// TwinCAT 3 PLC project Nepionic_Log_Klein
// Title: Nepionic_Log_Klein
// Company: Nepionic
// Author: Nepionic
// ProjectVersion: 0.1.0
// ProgramVersion: 3.1.4026.22
// libraries:
//   [Nepionic_Log], * (Nepionic)
//   Tc2_System, * (Beckhoff Automation GmbH)
//   Tc2_Utilities, * (Beckhoff Automation GmbH)
// project tree:
//   Lib/ KleinEventAppender.TcPOU, KleinEventEntry.TcDUT, KleinEventRing.TcDUT

// ---- Lib/KleinEventEntry.TcDUT
// One slot in the KleinEventRing.
//
// Binary layout (1280 bytes, little-endian, IDENTICAL in shape to
// Nepionic_Log_OTel.OTelLogEntry — see that type's doc comment. This is a
// deliberate reuse of the same proven wire layout under a new type name, not
// a coincidence: there is no reason to invent a different byte layout when
// this one is already implemented, tested, and documented on the Go side
// (github.com/siyka-au/klein, internal/receiver/ads/eventring.go). Giving it
// its own type name (rather than literally reusing OTelLogEntry) makes it an
// independently addressable ADS symbol under Nepionic_Log_Klein, decoupled
// from the deprecated Nepionic_Log_OTel library.
//
//   offset    0  ULINT   timestamp         Unix epoch nanoseconds
//   offset    8  UDINT   severity          0=Debug 1=Info 2=Warning 3=Error 4=Fatal
//                                            (raw PLC LogLevel ordinal — see the
//                                            PLC LogLevel -> Klein Severity mapping below)
//   offset   12  UDINT   attr_count        Number of populated entries in attrs (0..10)
//   offset   16  BYTE[192] message         STRING(191) null-terminated
//   offset  208  BYTE[64]  source          STRING(63)  null-terminated (instance path)
//   offset  272  BYTE[960] attrs           ARRAY[0..9] OF Nepionic_Log.LogAttribute (96 bytes each)
//                                            each attr:
//                                              offset  0  key         STRING(31)       = 32 bytes
//                                              offset 32  attr_type   LogAttributeType =  1 byte
//                                              offset 33  value_bytes ARRAY[0..62]     = 63 bytes
//   offset 1232  BYTE[44]  _pad
//   offset 1276  UDINT   sequence          ODD=being written, EVEN=committed (LAST field)
//   Total: 1280 bytes
//
// --- PLC LogLevel -> Klein Event mapping (Go: internal/receiver/ads/eventring.go) ---
//
// This is the precise mapping the Go decoder (KleinEventEntry -> model.Event)
// implements, documented here since no PLC toolchain was available in the
// authoring environment to verify it end-to-end against a live ring:
//
//   severity (raw UDINT, PLC LogLevel ordinal) -> model.Severity (klein/internal/model.Event.go):
//     0 (Debug)       -> SeverityDebug (2)
//     1 (Information) -> SeverityInfo  (3)
//     2 (Warning)     -> SeverityWarn  (4)
//     3 (Error)       -> SeverityError (5)
//     4 (Fatal)       -> SeverityFatal (6)
//     anything else   -> SeverityInfo  (3), clamped/defaulted (out-of-range raw value)
//
//   message   -> Event.Message                       (verbatim)
//   source    -> Event.Signal.Path                    (the resulting Event's identity)
//   source    -> Event.Actor.ID, with Event.Actor.Type fixed to "plc"
//               (a PLC-origin Event always carries a fixed Actor{Type: "plc", ID: source})
//   attrs[0..attr_count-1]
//             -> Event.To, as a model.StructValue{Fields: {attr.key: attr.value, ...}}
//                only when attr_count > 0 — an Event with no attributes leaves To nil
//                rather than emitting an empty Struct (Event has no dedicated
//                attributes field; To/From are otherwise unused by a pure
//                log-message Event, per docs/SPEC.md §9's "context lives either
//                as extra fields inside value's Struct, or in the sibling
//                attributes map" convention, adapted here since Event has no
//                sibling attributes map of its own).
//   timestamp -> Event.SourceTimestamp (int64 ns, direct copy)
{attribute 'pack_mode' := '1'}
TYPE KleinEventEntry :
STRUCT
	timestamp : ULINT;
	severity : UDINT;
	attribute_count : UDINT(0..10);
	message : STRING(191);
	source : STRING(63);
	attributes : ARRAY[0..9] OF Nepionic_Log.LogAttribute;
	_pad : ARRAY[0..43] OF BYTE;
	sequence : UDINT;
END_STRUCT
END_TYPE

// ---- Lib/KleinEventRing.TcDUT
// Ring buffer header + 128-slot event entry array.
// Exposed as an ADS symbol (e.g. MAIN.klein_appender.ring) and read by the Go
// Klein collector's ADS receiver (github.com/siyka-au/klein,
// internal/receiver/ads/eventring.go — DrainEvents/ParseEventSlot).
//
// Binary layout — IDENTICAL in shape to Nepionic_Log_OTel.OTelLogRing (same
// 64-byte header, same 128 x 1280-byte entries array). Deliberately reusing
// the proven ring-header layout under a new type name; see KleinEventEntry's
// doc comment for why.
//
//   offset  0  UDINT  head          Monotonically increasing write counter
//   offset  4  UDINT  capacity      Number of slots = 128
//   offset  8  UDINT  overflow_cnt  Incremented when ring is full
//   offset 12  UDINT  _reserved
//   offset 16  BYTE[48] _cache_pad  Pad header to 64 bytes
//   offset 64  KleinEventEntry[128] 128 x 1280 bytes = 163840 bytes
//   Total: 163904 bytes
TYPE KleinEventRing :
STRUCT
	head : UDINT;
	capacity : UDINT := 128;
	overflow_cnt : UDINT;
	_reserved : UDINT;
	_cache_pad : ARRAY[0..47] OF BYTE;
	entries : ARRAY[0..127] OF KleinEventEntry;
END_STRUCT
END_TYPE

// ---- Lib/KleinEventAppender.TcPOU
{attribute 'linkalways'}
{attribute 'no_explicit_call' := 'This FB is a CLASS and must be accessed using methods or properties'}
{attribute 'enable_dynamic_creation'}
/// Klein Event appender for Nepionic_Log.
/// Implements `LogAppender` by writing structured log entries directly into its
/// own `KleinEventRing` field (`ring`), which is exposed as an ADS symbol and
/// consumed by the Go Klein collector's ADS receiver
/// (github.com/siyka-au/klein, internal/receiver/ads/eventring.go), which
/// decodes each slot into a Klein `model.Event` — see KleinEventEntry.TcDUT's
/// doc comment for the exact severity/attribute/actor mapping.
///
/// The ring is owned by the appender — no external ring declaration is needed.
/// Just declare the appender in a PROGRAM or GVL so TwinCAT generates an ADS
/// symbol for it, then point the Klein collector's `ads` receiver at
/// `<PROGRAM>.<var_name>.ring` via an `event_rings` config entry.
///
/// This is the replacement for the deprecated `Nepionic_Log_OTel.OTelLogAppender`
/// (see that type's doc comment) — same seqlock ring-buffer pattern, same wire
/// shape, but decoded into a Klein `Event` instead of an OTel log record.
///
/// Usage:
/// ```st
/// // startup (e.g. MAIN FB_Init)
/// GetLogManager().Register(klein_appender);
///
/// // Klein ads receiver config:
/// //   event_rings:
/// //     - symbol: MAIN.klein_appender.ring
/// ```
FUNCTION_BLOCK PUBLIC KleinEventAppender IMPLEMENTS Nepionic_Log.LogAppender
VAR
	{attribute 'klein_role' := 'event_ring'}
	ring : KleinEventRing;
	_level : Nepionic_Log.LogLevel := Nepionic_Log.LogLevel.Debug;
END_VAR

METHOD PUBLIC Append : BOOL
VAR_INPUT
	level : Nepionic_Log.LogLevel;
	message : Tc2_System.T_MaxString;
	source : Tc2_System.T_MaxString;
	attributes : ARRAY[0..9] OF Nepionic_Log.LogAttribute;
	attribute_count : USINT;
END_VAR
VAR
	slot_idx : UDINT;
	expected_gen : UDINT;
	file_time : ULINT;
	i : USINT;
END_VAR
slot_idx := ring.head MOD ring.capacity;
expected_gen := (ring.head / ring.capacity + 1) * 2;

// Mark slot as being written (ODD sequence = write in progress)
ring.entries[slot_idx].sequence := expected_gen - 1;

// Timestamp — Windows FILETIME → Unix nanoseconds
file_time := Tc2_Utilities.F_GetSystemTime();
ring.entries[slot_idx].timestamp := (file_time - 116444736000000000) * 100;

// Severity — raw PLC LogLevel ordinal (0..4). Decoded on the Go side into
// model.Severity per the mapping documented in KleinEventEntry.TcDUT:
//   Debug=0 -> SeverityDebug(2), Information=1 -> SeverityInfo(3),
//   Warning=2 -> SeverityWarn(4), Error=3 -> SeverityError(5), Fatal=4 -> SeverityFatal(6).
CASE level OF
	Nepionic_Log.LogLevel.Debug:
		ring.entries[slot_idx].severity := 0;
	Nepionic_Log.LogLevel.Information:
		ring.entries[slot_idx].severity := 1;
	Nepionic_Log.LogLevel.Warning:
		ring.entries[slot_idx].severity := 2;
	Nepionic_Log.LogLevel.Error:
		ring.entries[slot_idx].severity := 3;
	Nepionic_Log.LogLevel.Fatal:
		ring.entries[slot_idx].severity := 4;
ELSE
	ring.entries[slot_idx].severity := 1;
END_CASE

// Payload — `source` becomes the resulting Klein Event's Signal.Path and
// Actor.ID (Actor.Type is fixed to "plc" on the Go side); `attributes`
// becomes the Event's To (a StructValue) when attribute_count > 0.
ring.entries[slot_idx].message := message;
ring.entries[slot_idx].source := source;
ring.entries[slot_idx].attribute_count := USINT_TO_UDINT(attribute_count);
FOR i := 0 TO 9 DO
	ring.entries[slot_idx].attributes[i] := attributes[i];
END_FOR

// Commit slot (EVEN sequence = ready for reader)
ring.entries[slot_idx].sequence := expected_gen;

// Increment overflow counter each time the write pointer wraps back to slot 0.
IF slot_idx = 0 AND ring.head > 0 THEN
	ring.overflow_cnt := ring.overflow_cnt + 1;
END_IF

// Advance write cursor
ring.head := ring.head + 1;

Append := TRUE;
END_METHOD

{attribute 'monitoring' := 'call'}
PROPERTY PUBLIC Level : Nepionic_Log.LogLevel
GET // PUBLIC
Level := _level;
END_GET
SET // PUBLIC
_level := Level;
END_SET
END_PROPERTY

END_FUNCTION_BLOCK
